// TIA Portal project "AIQS" (V18)

(* hardware
DEVICE "S7-1200-Station_1"  S7-1200 Station
   slot 0: "Baugruppenträger_0"  S7-1200 Rack  Rack  V1.0
   slot 1: "AIQS"  CPU 1215C DC/DC/DC  6ES7 215-1AG40-0XB0  V4.5
*)

// ===== PLC "AIQS"  CPU 1215C DC/DC/DC =====

VAR_GLOBAL   // PLC tag table "aiqs_steuer_variablen"
   "sauger_aussen" AT %I0.2 : Bool;   // DIa.2
   "encoder_A" AT %I0.3 : Bool;   // DIa.3
   "encoder_B" AT %I0.4 : Bool;   // DIa.4
   "sauger_innen" AT %I0.1 : Bool;   // DIa.1
   "eingang_LS" AT %I0.0 : Bool;   // DIa.0
   "sauger_rein" AT %Q0.0 : Bool;   // DQa.0
   "sauger_raus" AT %Q0.1 : Bool;   // DQa.1
   "band_rein" AT %Q0.2 : Bool;   // DQa.2
   "band_raus" AT %Q0.3 : Bool;   // DQa.3
   "kompressor" AT %Q0.4 : Bool;   // DQa.4
   "sauger_PWM" AT %Q0.6 : Bool;   // DQa.6
   "band_PWM" AT %Q0.7 : Bool;   // DQa.7
   "sauger_runter" AT %Q1.0 : Bool;   // DQb.0
   "ventil_Vakuum" AT %Q1.1 : Bool;   // DQb.1
END_VAR

DATA_BLOCK "DB_Ablauf"   // DB1
{ S7_Optimized_Access := 'TRUE' }
VERSION : 0.1
// stored: InstanceOfName FB_Ablauf
"FB_Ablauf"
BEGIN
END_DATA_BLOCK

DATA_BLOCK "DB_Referenzen"   // DB2
{ S7_Optimized_Access := 'TRUE' }
VERSION : 0.1
   VAR RETAIN
      Calib : Struct
         zeitKamera : Time := T#745MS;
         zeitAusschuss : Time := T#1S;
         zeitProzessEnde : Time := T#2S;   // Zeit bevor die ProzessEnde Flag in der OPCUA-Schnittstelle gesetzt wird
         zeitMitteLS : Time := T#20MS;   // Zeit die das Band weiterfährt um das WP mittig in der Lichtschranke zu positionieren
         zeit_saugerRunter : Time := T#700MS;   // Zeit die der Sauger nach unten gedrückt wird und dort verharrt
         zeit_vakuumloesen : Time := T#200MS;   // Zeit die gewartet wird um dem Saugnapf die möglichkeit zu geben sich zu lösen
         zeitVorFoto : Time := T#500MS;
         zeitVorFehlercheck : Time := T#500MS;   // Zeit die vor dem Fehlercheck die nach dem PICK gewartet wird
         zeitVakuumErzeugen : Time := T#200MS;   // Zeit für den Kompressor Vakuum aufzubauen
      END_STRUCT;
      Defaults : Struct
         zeitKamera : Time := T#745MS;
         zeitAusschuss : Time := T#1S;
         zeitProzessEnde : Time := T#2S;
         zeitMitteLS : Time := T#20MS;
         zeitVorFoto : Time := T#500MS;
         zeit_saugerRunter : Time := T#700MS;
         zeit_vakuumloesen : Time := T#200MS;
         zeitVorFehlercheck : Time := T#500MS;
         zeitVakuumErzeugen : Time := T#200MS;
      END_STRUCT;
   END_VAR
BEGIN
END_DATA_BLOCK

DATA_BLOCK "FB_Kalibrierung_DB"   // DB3
{ S7_Optimized_Access := 'TRUE' }
VERSION : 0.1
// stored: InstanceOfName FB_Kalibrierung
"FB_Kalibrierung"
BEGIN
END_DATA_BLOCK

DATA_BLOCK "DB_Version"   // DB4
{ S7_Optimized_Access := 'TRUE' }
VERSION : 0.1
   VAR
      "version" : String := '1.3.0';
   END_VAR
BEGIN
END_DATA_BLOCK

FUNCTION_BLOCK "FB_Ablauf"   // FB1, SCL
{ S7_Optimized_Access := 'TRUE' }
VERSION : 0.1
   VAR RETAIN
      modell : String := 'AIQS';
   END_VAR
   VAR
      idle : Bool;
      pick : Bool;
      drop : Bool;
      good : Bool;
      bad : Bool;
      Kalibrierung : Struct
         KALIBRIERE : Bool;
         kalibAktiv : Bool;
         BEENDEN : Bool;
         Kalibriere_finished : Bool;
         DEFAULT : Bool;
         default_finished : Bool;
         FAHRE_VOR : Bool;
         fahrZeit : Time;
         fahre_finished : Bool;
         FAHRE_ZURUECK : Bool;
         zurueck_finished : Bool;
         FAHRE_ZURUECK_KURZ : Bool;
         zurueck_kurz_finished : Bool;
      END_STRUCT;
      pick_finished : Bool;
      drop_finished : Bool;
      good_finished : Bool;
      bad_finished : Bool;
      warte_start : Bool;
      warte_zeit : Time := T#500ms;
      "step" : Int;
      warte : TON_TIME;
      pick_failed : Bool;
      move_to_camera : Bool;
      move_to_camera_finished : Bool;
      drop_failed : Bool;
      drop_aktiv : Bool;
      pick_aktiv : Bool;
      good_aktiv : Bool;
      bad_aktiv : Bool;
      move_to_camera_aktiv : Bool;
   END_VAR
BEGIN
   #warte.TON(IN := #warte_start, PT := #warte_zeit);

   // Stepchain AIQS
   CASE #step OF
       0: // init
           #modell := 'AIQS';
           #step := 1;
       1: // reset
           #bad_finished := FALSE;
           #good_finished := FALSE;
           #move_to_camera_finished := FALSE;
           #Kalibrierung.Kalibriere_finished := FALSE;
           #drop_failed := FALSE;
           #drop_finished := FALSE;
           #pick_finished := FALSE;
           #pick_failed := FALSE;
           #idle := TRUE;
           #step := 2
           ;
       2: // Fallunterscheidung
           IF #pick THEN
               #pick_aktiv := TRUE;
               #pick := FALSE;
               #idle := FALSE;
               #step := 10;
           ELSIF #drop THEN
               #drop_aktiv := TRUE;
               #drop := FALSE;
               #idle := FALSE;
               #step := 30;
           ELSIF #move_to_camera THEN
               #move_to_camera_aktiv := TRUE;
               #move_to_camera := FALSE;
               #idle := FALSE;
               #step := 50;
           ELSIF #good THEN
               #good_aktiv := TRUE;
               #good := FALSE;
               #idle := FALSE;
               #step := 60;
           ELSIF #bad THEN
               #bad_aktiv := TRUE;
               #bad := FALSE;
               #idle := FALSE;
               #step := 70;
           ELSIF #Kalibrierung.KALIBRIERE THEN
               #Kalibrierung.KALIBRIERE := FALSE;
               #Kalibrierung.kalibAktiv := TRUE;
               #idle := FALSE;
               #step := 100;
           END_IF
           ;

       200: // Ende jedes Prozesses
           "band_PWM" := FALSE;
           "band_raus" := FALSE;
           "band_rein" := FALSE;
           "sauger_PWM" := FALSE;
           "sauger_raus" := FALSE;
           "sauger_rein" := FALSE;
           #warte_zeit := "DB_Referenzen".Calib.zeitProzessEnde;
           #warte_start := TRUE;
           IF #warte.Q THEN
               #warte_start := FALSE;
               #step := 1;
           END_IF
           ;

       10: //  -------------------------------------------------------------------  PICK Start
           "sauger_PWM" := TRUE;
           #step := 11;
       11: // sauger raus bis schalter
           "sauger_raus" := TRUE;
           IF "sauger_aussen" THEN
               "sauger_raus" := FALSE;
               #step := 13;
           END_IF
           ;
       13: // kurz warten
           #warte_start := TRUE;
           #warte_zeit := T#200ms;
           IF #warte.Q THEN
               #warte_start := FALSE;
               #step := 14;
           END_IF;
       14: // Sauger nimmt WP auf
           "kompressor" := TRUE;
           #step := 15;
       15: // warten auf Druckaufbau
           #warte_start := TRUE;
           #warte_zeit := "DB_Referenzen".Calib.zeitVakuumErzeugen;
           IF #warte.Q THEN
               #warte_start := FALSE;
               #step := 16;
           END_IF;
       16: // saugerkopf nach unten
           "sauger_runter" := TRUE;
           #step := 17;
       17: // Saugerkopf aktivieren
           #warte_zeit := "DB_Referenzen".Calib.zeit_saugerRunter;
           #warte_start := TRUE;
           IF #warte.Q THEN
               "ventil_Vakuum" := TRUE;
               #warte_start := FALSE;
               #step := 18;
           END_IF
           ;
       18: // saugerkopf nach oben
           #warte_zeit := "DB_Referenzen".Calib.zeitVakuumErzeugen;
           #warte_start := TRUE;
           IF #warte.Q THEN
               #warte_start := FALSE;
               "sauger_runter" := FALSE;
               #step := 19;
           END_IF
           ;
       19: // Sauger fährt rein
           "sauger_rein" := TRUE;
           IF "sauger_innen" THEN
               "sauger_rein" := FALSE;
               #step := 21;
           END_IF
           ;
       21: // Saugerkopf deaktivieren
           "sauger_runter" := TRUE;
           #warte_zeit := "DB_Referenzen".Calib.zeit_saugerRunter;
           #warte_start := TRUE;
           IF #warte.Q THEN
               #warte_start := FALSE;
               "ventil_Vakuum" := FALSE;
               #step := 22;
           END_IF
           ;
       22: // aus
           #warte_zeit := "DB_Referenzen".Calib.zeit_vakuumloesen;
           #warte_start := TRUE;
           IF #warte.Q THEN
               "sauger_runter" := FALSE;
               "kompressor" := FALSE;
               #step := 23;
           END_IF
           ;
       23: //  warten vor Fehlercheck
           #warte_start := TRUE;
           #warte_zeit := "DB_Referenzen".Calib.zeitVorFehlercheck;
           IF #warte.Q THEN
               #warte_start := FALSE;
               #step := 24;
           END_IF
           ;
       24: // checken ob WP jetzt auf band und Ende
           IF "eingang_LS" THEN
               #pick_failed := TRUE;
           ELSE
               #pick_finished := TRUE;
           END_IF;
           #pick_aktiv := FALSE;
           #step := 200;
           //  ------------------------------------------------------------------- ENDE PICK
       50: //  ------------------------------------------------------------------- START Move to camera
           "band_PWM" := TRUE;
           #step := 51;
       51: // band rein bis unter camera
           "band_raus" := FALSE;
           "band_rein" := TRUE;
           #warte_zeit := "DB_Referenzen".Calib.zeitKamera;
           #warte_start := TRUE;
           IF #warte.Q THEN
               #warte_start := FALSE;
               "band_rein" := FALSE;
               #step := 52;
           END_IF
           ;
       52: // ENDE
           #move_to_camera_aktiv := FALSE;
           #warte_zeit := "DB_Referenzen".Calib.zeitVorFoto;
           #warte_start := TRUE;
           IF #warte.Q THEN
               #warte_start := FALSE;
               #move_to_camera_finished := TRUE;
               #step := 200;
           END_IF
           ;
           //  ------------------------------------------------------------------- ENDE Move to Camera
       60: //  ------------------------------------------------------------------- START good
           "band_PWM" := TRUE;
           "band_raus" := TRUE;
           IF NOT "eingang_LS" THEN
               #step := 61;
           END_IF;
       61: // mittig unter den saugkopf fahren
           #warte_start := TRUE;
           #warte_zeit := "DB_Referenzen".Calib.zeitMitteLS;
           IF #warte.Q THEN
               #warte_start := FALSE;
               "band_raus" := FALSE;
               "band_PWM" := FALSE;
               #good_aktiv := FALSE;
               #good_finished := TRUE;
               #step := 200;
           END_IF;
           //  ------------------------------------------------------------------- ENDE good
       70: //  ------------------------------------------------------------------- START bad
           "band_PWM" := TRUE;
           "band_rein" := TRUE;
           #warte_start := TRUE;
           #warte_zeit := "DB_Referenzen".Calib.zeitAusschuss;
           IF #warte.Q THEN
               #warte_start := FALSE;
               #step := 71;
           END_IF
           ;
       71: // Ausmachen
           "band_rein" := FALSE;
           "band_PWM" := FALSE;
           #bad_aktiv := FALSE;
           #bad_finished := TRUE;
           #step := 200;
           //  ------------------------------------------------------------------- ENDE bad
       30: //  ------------------------------------------------------------------- START drop
           "sauger_PWM" := TRUE;
           #step := 31;
       31: // sauger rein bis schalter "sauger_innen"
           "sauger_rein" := TRUE;
           IF "sauger_innen" THEN
               "sauger_rein" := FALSE;
               #step := 34;
           END_IF;
       34: // Sauger nimmt WP auf
           "kompressor" := TRUE;
           #step := 36;
       36: // saugerkopf nach unten
           "sauger_runter" := TRUE;
           #step := 37;
       37: // Saugerkopf aktivieren
           #warte_start := TRUE;
           #warte_zeit := "DB_Referenzen".Calib.zeit_saugerRunter;
           IF #warte.Q THEN
               "ventil_Vakuum" := TRUE;
               #warte_start := FALSE;
               #step := 38;
           END_IF;
       38: // saugerkopf nach oben nach Vakuum erzeugen
           #warte_start := TRUE;
           #warte_zeit := "DB_Referenzen".Calib.zeitVakuumErzeugen;
           IF #warte.Q THEN
               "sauger_runter" := FALSE;
               #warte_start := FALSE;
               #step := 39;
           END_IF
           ;
       39: // sauger raus
           "sauger_raus" := TRUE;
           IF "sauger_aussen" THEN
               "sauger_raus" := FALSE;
               #step := 42;
           END_IF;
       42: // saugerkopf nach unten
           "sauger_runter" := TRUE;
           #step := 43;
       43: // Saugerkopf deaktivieren
           #warte_zeit := "DB_Referenzen".Calib.zeit_saugerRunter;
           #warte_start := TRUE;
           IF #warte.Q THEN
               "ventil_Vakuum" := FALSE;
               #warte_start := FALSE;
               #step := 44;
           END_IF;
       44: // kompressor aus
           #warte_zeit := "DB_Referenzen".Calib.zeit_vakuumloesen;
           #warte_start := TRUE;
           IF #warte.Q THEN
               #warte_start := FALSE;
               "kompressor" := FALSE;
               #step := 45;
           END_IF;

       45: // saugerkopf nach oben
           "sauger_runter" := FALSE;
           #step := 46;
       46: // sauger rein bis schalter
           "sauger_rein" := TRUE;
           IF "sauger_innen" THEN
               "sauger_rein" := FALSE;
               #step := 48;
           END_IF
           ;
       48: // Check ob Failed und ENDE
           IF NOT "eingang_LS" THEN
               #drop_failed := TRUE;
           ELSE 
               #drop_finished := TRUE;
           END_IF;
           #drop_aktiv := FALSE;
           #step := 200;
           // ------------------------------------------------------------------- ENDE DROP
       100: // warte auf ende Kalibrierung
           #pick := FALSE;
           #drop := FALSE;
           #bad := FALSE;
           #good := FALSE;
           #move_to_camera := FALSE;
           IF NOT #Kalibrierung.kalibAktiv AND #Kalibrierung.Kalibriere_finished THEN
               #step := 200;
           END_IF
           ;
       ELSE
           ;
   END_CASE;
END_FUNCTION_BLOCK

FUNCTION_BLOCK "FB_Kalibrierung"   // FB2, FBD
{ S7_Optimized_Access := 'TRUE' }
VERSION : 0.1
   VAR
      "step" : DInt;
      Warten : TON_TIME;
      warteStart : Bool;
      warteZeit : Time;
   END_VAR
BEGIN

REGION Network 1 (SCL): Ablauf Kalibrierung
   CASE #step OF
       0:  // Init
           "DB_Ablauf".Kalibrierung.DEFAULT := FALSE;
           "DB_Ablauf".Kalibrierung.BEENDEN := FALSE;
           "DB_Ablauf".Kalibrierung.FAHRE_VOR := FALSE;
           "DB_Ablauf".Kalibrierung.FAHRE_ZURUECK := FALSE;
           IF "DB_Ablauf".Kalibrierung.kalibAktiv THEN
               #step := 1;
           END_IF
           ;
       1: // Warten auf Befehle
           IF "DB_Ablauf".Kalibrierung.DEFAULT THEN
               "DB_Ablauf".Kalibrierung.DEFAULT := FALSE;
               #step := 100;
           ELSIF "DB_Ablauf".Kalibrierung.BEENDEN THEN
               "DB_Ablauf".Kalibrierung.BEENDEN := FALSE;
               #step := 90;
           ELSIF "DB_Ablauf".Kalibrierung.FAHRE_VOR THEN
               "DB_Ablauf".Kalibrierung.FAHRE_VOR := FALSE;
               #step := 20;
           ELSIF "DB_Ablauf".Kalibrierung.FAHRE_ZURUECK THEN
               "DB_Ablauf".Kalibrierung.FAHRE_ZURUECK := FALSE;
               #step := 50;
           END_IF
           ;

       20: // Power auf Motor
           "band_PWM" := TRUE;
           "band_raus" := FALSE;
           "band_rein" := FALSE;
           #step := 21;
       21: // WP von Eingang (Position nach PICK) Richtung Kamera mit mitgelieferter Zeit
           "band_raus" := FALSE;
           "band_rein" := TRUE;
           #warteZeit := "DB_Ablauf".Kalibrierung.fahrZeit;
           #warteStart := TRUE;
           IF #Warten.Q THEN
               #warteStart := FALSE;
               "band_raus" := FALSE;
               "band_rein" := FALSE;
               #step := 22;
           END_IF
           ;
       22: // Fahre finished
           "band_PWM" := FALSE;
           "band_raus" := FALSE;
           "band_rein" := FALSE;

           "DB_Ablauf".Kalibrierung.fahre_finished := TRUE;
           #warteZeit := "DB_Referenzen".Calib.zeitProzessEnde;
           #warteStart := TRUE;
           IF #Warten.Q THEN
               "DB_Ablauf".Kalibrierung.fahre_finished := FALSE;
               #warteStart := FALSE;
               #step := 0;
           END_IF
           ;

       50: // Power auf Motor
           "band_PWM" := TRUE;
           "band_raus" := FALSE;
           "band_rein" := FALSE;

           #step := 51
           ;
       51: // rausfahren bis WP an Lichtschranke
           "band_raus" := TRUE;
           "band_rein" := FALSE;
           #warteZeit := "DB_Ablauf".Kalibrierung.fahrZeit;
           #warteStart := TRUE;
           IF NOT "eingang_LS" OR #Warten.Q THEN
               #warteStart := FALSE;
               "band_raus" := FALSE;
               "band_rein" := FALSE;
               #step := 52;
           END_IF
           ;
       52: // kurz warten
           "DB_Ablauf".Kalibrierung.zurueck_finished := TRUE;
           #warteZeit := "DB_Referenzen".Calib.zeitProzessEnde;
           #warteStart := TRUE;
           IF #Warten.Q THEN
               "DB_Ablauf".Kalibrierung.zurueck_finished := FALSE;
               #warteStart := FALSE;
               #step := 0;
           END_IF
           ;
       70: // unter sauger fahren
           "band_raus" := TRUE;
           "band_rein" := FALSE;
           #warteZeit := "DB_Ablauf".Kalibrierung.fahrZeit;
           #warteStart := TRUE;
           IF #Warten.Q THEN
               "band_raus" := FALSE;
               "band_rein" := FALSE;
               #warteStart := FALSE;
               #step := 71;
           END_IF
           ;
       71: // kurz warten
           "DB_Ablauf".Kalibrierung.zurueck_kurz_finished:= TRUE;
           #warteZeit := "DB_Referenzen".Calib.zeitProzessEnde;
           #warteStart := TRUE;
           IF #Warten.Q THEN
               "DB_Ablauf".Kalibrierung.zurueck_kurz_finished := FALSE;
               #warteStart := FALSE;
               #step := 0;
           END_IF
           ;
       90: // Kalibrierung Beenden
           "DB_Ablauf".Kalibrierung.kalibAktiv := FALSE;
           "DB_Ablauf".Kalibrierung.Kalibriere_finished := TRUE;
           #step := 0
           ;
       100: // Auf default zurücksetzen
           "DB_Referenzen".Calib.zeitKamera := "DB_Referenzen".Defaults.zeitKamera;
           "DB_Referenzen".Calib.zeitAusschuss := "DB_Referenzen".Defaults.zeitAusschuss;
           "DB_Referenzen".Calib.zeitProzessEnde := "DB_Referenzen".Defaults.zeitProzessEnde;
           "DB_Referenzen".Calib.zeitMitteLS := "DB_Referenzen".Defaults.zeitMitteLS;
           "DB_Referenzen".Calib.zeit_saugerRunter := "DB_Referenzen".Defaults.zeit_saugerRunter;
           "DB_Referenzen".Calib.zeitVorFoto := "DB_Referenzen".Defaults.zeitVorFoto;
           "DB_Referenzen".Calib.zeit_vakuumloesen := "DB_Referenzen".Defaults.zeit_vakuumloesen;

           #step := 101
           ;
       101: // default finished
           "DB_Ablauf".Kalibrierung.default_finished := TRUE;
           #warteStart := TRUE;
           #warteZeit := "DB_Referenzen".Calib.zeitProzessEnde;
           IF #Warten.Q THEN
               #warteStart := FALSE;
               "DB_Ablauf".Kalibrierung.default_finished := FALSE;
               #step := 1;
           END_IF
           ;

       ELSE  // Statement section ELSE
           ;
   END_CASE;
END_REGION

REGION Network 2
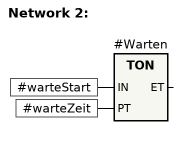
   #Warten(IN := #warteStart, PT := #warteZeit);   // TON
END_REGION
END_FUNCTION_BLOCK

ORGANIZATION_BLOCK "Main"   // OB1, FBD, ProgramCycle
TITLE = "Main Program Sweep (Cycle)"
{ S7_Optimized_Access := 'TRUE' }
VERSION : 0.1
   VAR_INPUT
      Initial_Call : Bool;   // Initial call of this OB
      Remanence : Bool;   // =True, if remanent data are available
   END_VAR
BEGIN

REGION Network 1
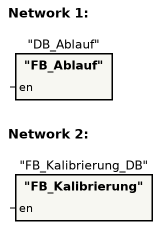
   "DB_Ablauf"();   // "FB_Ablauf"
END_REGION

REGION Network 2
   "FB_Kalibrierung_DB"();   // "FB_Kalibrierung"
END_REGION
END_ORGANIZATION_BLOCK